Fanuc KAREL source: ko00031.KL

PROGRAM KO00031
%STACKSIZE=65535
%PRIORITY=65535
%NOLOCKGROUP
VAR
P1 : JOINTPOS9
P2 : JOINTPOS9
P3 : JOINTPOS9
P4 : JOINTPOS9
OUT : XYZWPREXT
BEGIN
-- UNRESOLVED_PC line 10 opcodes [27 27 49 7E AD 27 49 7E AD 27 49 7E AD 27 49 7E AD 76 7E 4A] marker_code=0
END KO00031
